{attribute 'qualified_only'}
VAR_GLOBAL
	Logger		: SimpleLog<2>;
END_VAR

(* stored: Version 1.1.0.1
   GVL GVL: Id {3d40af9c-14b4-45f5-a52a-73f347280f7c} *)
